FUNCTION_BLOCK "ST10_StopperCtrl"
VAR
  Stopper : Array[1..100] of "StopperCtrl";
END_VAR
BEGIN
  // Původní jazyk: LAD
  // Zdroj XML: EXPORT/Program blocks/OP010/10_Device/26_Stopper/ST10_StopperCtrl.xml
  // (Žádný StructuredText network nebyl nalezen; LAD/STL/GRAPH není automaticky překládán.)
END_FUNCTION_BLOCK
